FUNCTION_BLOCK DSCYL_SVR (* Double-Stroke Cylinder Server for a Remote DSCYL_PRXY *)
  (* Standard: 61499-1 *)
  (* Version 0.0, 2004-09-26, JHC, Rockwell Automation, Adapted from DSCYL_MDL1. *)
  (* Compiler header: package fb.rt.mach; import fb.rt.net.*; *)
  (* Compiler Java Sun JDK 1.4.2 *)
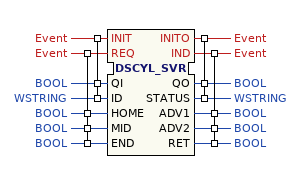
  EVENT_INPUT
    INIT WITH QI, ID; (* Initialize Server *)
    REQ WITH HOME, MID, END; (* Send Sensor Data *)
  END_EVENT
  EVENT_OUTPUT
    INITO WITH QO, STATUS; (* INIT Acknowledgment *)
    IND WITH ADV1, ADV2, RET; (* Actuator Change Indication *)
  END_EVENT
  VAR_INPUT
    QI : BOOL; (* Event Input Qualifier *)
    ID : WSTRING; (* Connection Identifier *)
    HOME : BOOL; (* Both cylinders HOME *)
    MID : BOOL; (* CYL1 at END,CYL2 HOME *)
    END : BOOL; (* Both cylinders at END *)
  END_VAR
  VAR_OUTPUT
    QO : BOOL; (* Event Output Qualifier *)
    STATUS : WSTRING; (* Service Status *)
    ADV1 : BOOL; (* ADVANCE Cyl#1 *)
    ADV2 : BOOL; (* ADVANCE Cyl#2 *)
    RET : BOOL; (* RETRACT Both Cylinders *)
  END_VAR
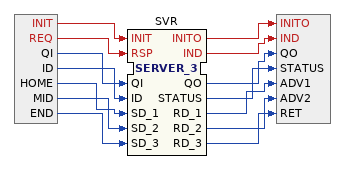
  FBS
    SVR : SERVER_3;
  END_FBS
  EVENT_CONNECTIONS
    INIT TO SVR.INIT;
    SVR.INITO TO INITO;
    REQ TO SVR.RSP;
    SVR.IND TO IND;
  END_CONNECTIONS
  DATA_CONNECTIONS
    QI TO SVR.QI;
    SVR.QO TO QO;
    ID TO SVR.ID;
    SVR.STATUS TO STATUS;
    HOME TO SVR.SD_1;
    MID TO SVR.SD_2;
    END TO SVR.SD_3;
    SVR.RD_1 TO ADV1;
    SVR.RD_2 TO ADV2;
    SVR.RD_3 TO RET;
  END_CONNECTIONS
END_FUNCTION_BLOCK
